PROGRAM task21
VAR
	stTimer2 : ST_Timer := (myTime := T#5S);
	fbTimeOff : TOF := (PT := stTimer2.myTime);
END_VAR

fbTimeOff(IN := stTimer2.myBool);

END_PROGRAM

(* stored: Version 1.1.0.1, ProductVersion 3.1.4024.12
   POU task21: Id {ab5dd975-8dc7-4f37-ad54-5afc1194300e}, SpecialFunc None *)
